(* CODESYS project OOP-test_with_lib.ecp

Project tree, tasks and I/O mapping:
  GenericDummyMasterDevice : Generic Master, WAGO Automation, order no. None, version 1.0.0.0
  PFC200_CS_2ETH_CAN : 750-8203 PFC200 2ETH CAN, WAGO, order no. 0750-8203, version 1.3.1.33
    application Application
      libraries: ; CoDeSys Library Template Interfaces, * (3S - Smart Software Solutions GmbH); VisuDialogs, * (System)
      task PLC_Task (cyclic, interval t#10ms, priority 14) calls PLC_PRG
      task VISU_TASK (cyclic, interval 100 ms, priority 15) calls VisuElems.Visu_Prg
      program PLC_PRG [ST]
      visualisation Visualization
      visualisation Visualization_1
    DeviceAdapter
    Kbus : Kbus, WAGO, version 1.1.0.1
        settings: k-bus event control 1.offset = 1
        unmapped channels: K-BUS diagnostics
      _4_DO_24_V_DC_0_5A_4_Bit_Diag : 0750-0532, WAGO, order no. 0750-0532, version 0.0.0.9
          settings: K-BUS Module slot index = 2
          output R1_l1 : BOOL  // _OUT._OUT
          output R2L1 : BOOL  // _OUT._OUT
          output R2_L2 : BOOL  // _OUT._OUT
          unmapped channels: _IN, _OUT
        DeviceAdapter
      _4_DI_24_V_DC_3_0ms : 0750-0432, WAGO, order no. 0750-0432, version 0.0.0.9
          settings: K-BUS Module slot index = 1
          unmapped channels: _IN
        DeviceAdapter
      RS_232_RS_485_Interface_adjustable : 0750-0652, WAGO, order no. 0750-0652, version 0.0.0.22
          settings: K-BUS Module slot index = 3
          unmapped channels: _INPUTCHANNEL, _OUTPUTCHANNEL
        DeviceAdapter
      _4_AI_4_20mA_s_e : 0750-0455, WAGO, order no. 0750-0455, version 0.0.0.10
          settings: K-BUS Module slot index = 4
          unmapped channels: _IW 1, _IW 2, _IW 3, _IW 4
        DeviceAdapter
    MODBUS
      MODBUS : MODBUS, WAGO, order no. n/a, version 1.1.1.11
    CANbus
      WAGO_CANopen_Local_Device : WAGO CANopen Device, WAGO, version 3.5.3.9
  text list GlobalTextList
  global variables Global_Variable
*)

// Global_Variable
VAR_GLOBAL
	myTime AT%MW1: WORD :=0;
	Day AT%MW0: BOOL := TRUE;	

END_VAR

// PFC200_CS_2ETH_CAN/Application/PLC_PRG
PROGRAM PLC_PRG
VAR
	r1: SNT.RoomType1;
	r2: SNT.RoomType2;
	r3: SNT.RoomType3;
	
	Rooms: ARRAY [1..k] OF SNT.IRoom:=[r1,r2,r3];
	i:INT;
	
	timer_my: INT :=0;
END_VAR
VAR CONSTANT
	k: INT :=3;
	
END_VAR

// test of github
FOR i:=1 TO k DO 
	myTime := myTime + 1;
	IF NOT Day THEN 
		Rooms[i].OperationDay();
		ELSE
		Rooms[i].OperationNight();
	END_IF
	R1_l1 := Day;
END_FOR

IF myTime < 750 THEN
	Day := TRUE;
	ELSE 
	Day := FALSE;		
END_IF


IF myTime> 1500 THEN
	myTime :=0;
END_IF

END_PROGRAM

// PFC200_CS_2ETH_CAN/Application/Visualization
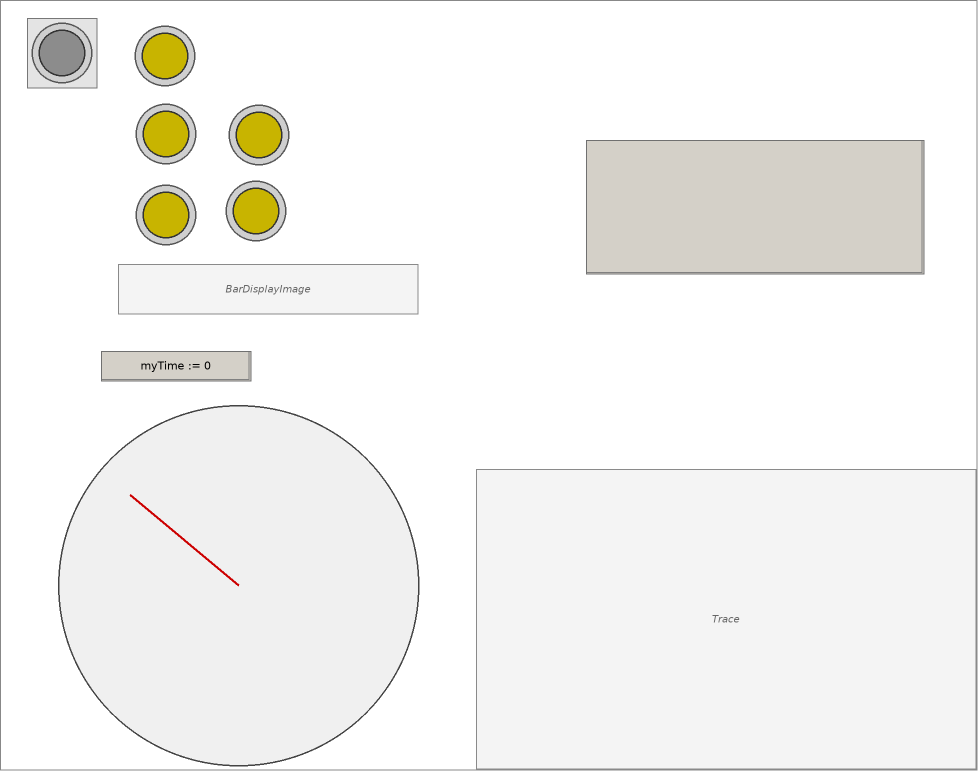
VISUALIZATION Visualization  // 978x771
VAR_IN_OUT
END_VAR
VAR
	bResetTrigger : BOOL;
	bStart : BOOL;
	bStop : BOOL;
END_VAR
    Lamp1 (130,21 70x70), variable: PLC_PRG.r1.bLight, style: Lamp-Lamp1-Yellow
    Lamp1 (131,99 70x70), variable: PLC_PRG.r2.bLight, style: Lamp-Lamp1-Yellow
    Lamp1 (224,100 70x70), variable: PLC_PRG.r2.bAddLight, style: Lamp-Lamp1-Yellow
    Lamp1 (131,180 70x70), variable: PLC_PRG.r3.bLight, style: Lamp-Lamp1-Yellow
    Lamp1 (221,176 70x70), variable: PLC_PRG.r3.bAddLight, style: Lamp-Lamp1-Yellow
    PushSwitchLed (27,18 70x70), variable: Day, behaviour: TOGGLE, style: Switch-PushSwitchLed-Gray
    BarDisplayImage (118,264 300x50), value: PLC_PRG.r3.iTemp, style: BarDisplayImage-Gray, scale format: %.0f, scale 15..30
    Meter360 (27,405 423x361), value: myTime, style: Meter-Meter360-Gray, scale format: %.0f, scale 0..1500
    Button (101,351 150x30), "myTime := 0"
        OnMouseClick: execute { myTime:=0; }
    Trace (476,469 500x300)
    Button (586,140 338x134)
        OnMouseClick:  Assign=Visualization_1, Type=Assignment
        OnMouseDown:  Assign=Visualization_1, Type=Assignment
END_VISUALIZATION

// PFC200_CS_2ETH_CAN/Application/Visualization_1
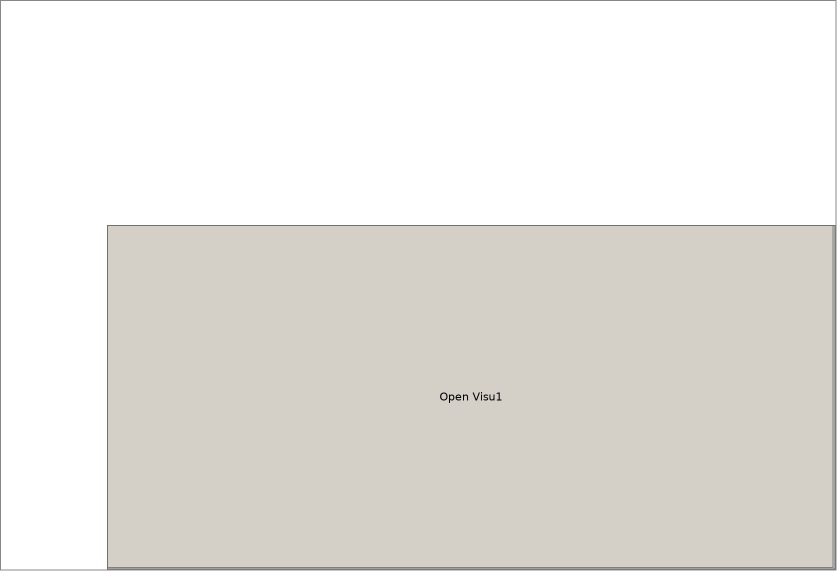
VISUALIZATION Visualization_1  // 837x571
    Button (107,225 728x344), "Open Visu1"
        OnMouseClick:  Type=Previous
END_VISUALIZATION
